{attribute 'qualified_only'}
{attribute 'strict'}
{attribute 'to_string'}
TYPE E_EventReaction :
(
	Undefined 			:= 0,
	NoReaction 			:= 1,
	CycleStop			:= 11,
	Stop 				:= 21,
	Init				:= 31
);
END_TYPE

(* stored: Version 1.1.0.1
   DUT E_EventReaction: Id {553040c7-0eeb-48c9-a147-5daf2b6b606f} *)
